// TIA Portal V18 export
FUNCTION_BLOCK "productionCounter"   // FB8, FBD
{ S7_Optimized_Access := 'TRUE' }
// stored: MemoryReserve 100, SetENOAutomatically false
   VAR_INPUT
      I_partProduced : Bool;
      I_nokPart : Bool;
   END_VAR
   VAR_IN_OUT
      IO_actualValues : "UDT_actualValues";
      IO_PreviousValues : "UDT_actualValues";
      IO_settings : "UDT_settings";
      IO_control : "UDT_control";
      IO_settingsShift1 : "UDT_settingsShift";
      IO_settingsShift2 : "UDT_settingsShift";
      IO_settingsShift3 : "UDT_settingsShift";
      IO_locTime : DTL;
   END_VAR
   VAR
      fpBit_resetCounters : Bool;
      fpBit_partProduced : Bool;
      fpBit_nokPart : Bool;
      fpBit_stop : Bool;
      fpBit_start : Bool;
      RS_taktTimeEn : Bool;
      TIM_taktTime { S7_SetPoint := 'True'} : TONR_TIME;
      memTaktTime : DInt;
      shiftTrigger0 { S7_SetPoint := 'True'} : "shiftTrigger";
      shiftTrigger1 { S7_SetPoint := 'True'} : "shiftTrigger";
      shiftTrigger2 { S7_SetPoint := 'True'} : "shiftTrigger";
      TaktTimeElapsed { S7_SetPoint := 'True'} : Time;
   END_VAR
   VAR_TEMP
      T_resetTaktTimeTimer : Bool;
      T_changeTaktTimeTimer : Bool;
      T_actualTOD : Time_Of_Day;
      T_shiftTrigger : Array[0..2] of Struct
         active : Bool;
         taktTimeEn : Bool;
         startDetect : Bool;
      END_STRUCT;
      T_control : Struct
         stop : Bool;
         start : Bool;
         resetCounters : Bool;
         taktTimeEn : Bool;
      END_STRUCT;
      T_settings : Struct
         enabled : Bool;
         autostartEnabled : Bool;
      END_STRUCT;
   END_VAR
   VAR_TEMP   // added for the SCL form of the ladder/FBD networks
      _w1 : Bool;
   END_VAR
BEGIN

REGION Network 1: free
END_REGION

REGION Network 2: actual TOD / Convert actual local time to TOD
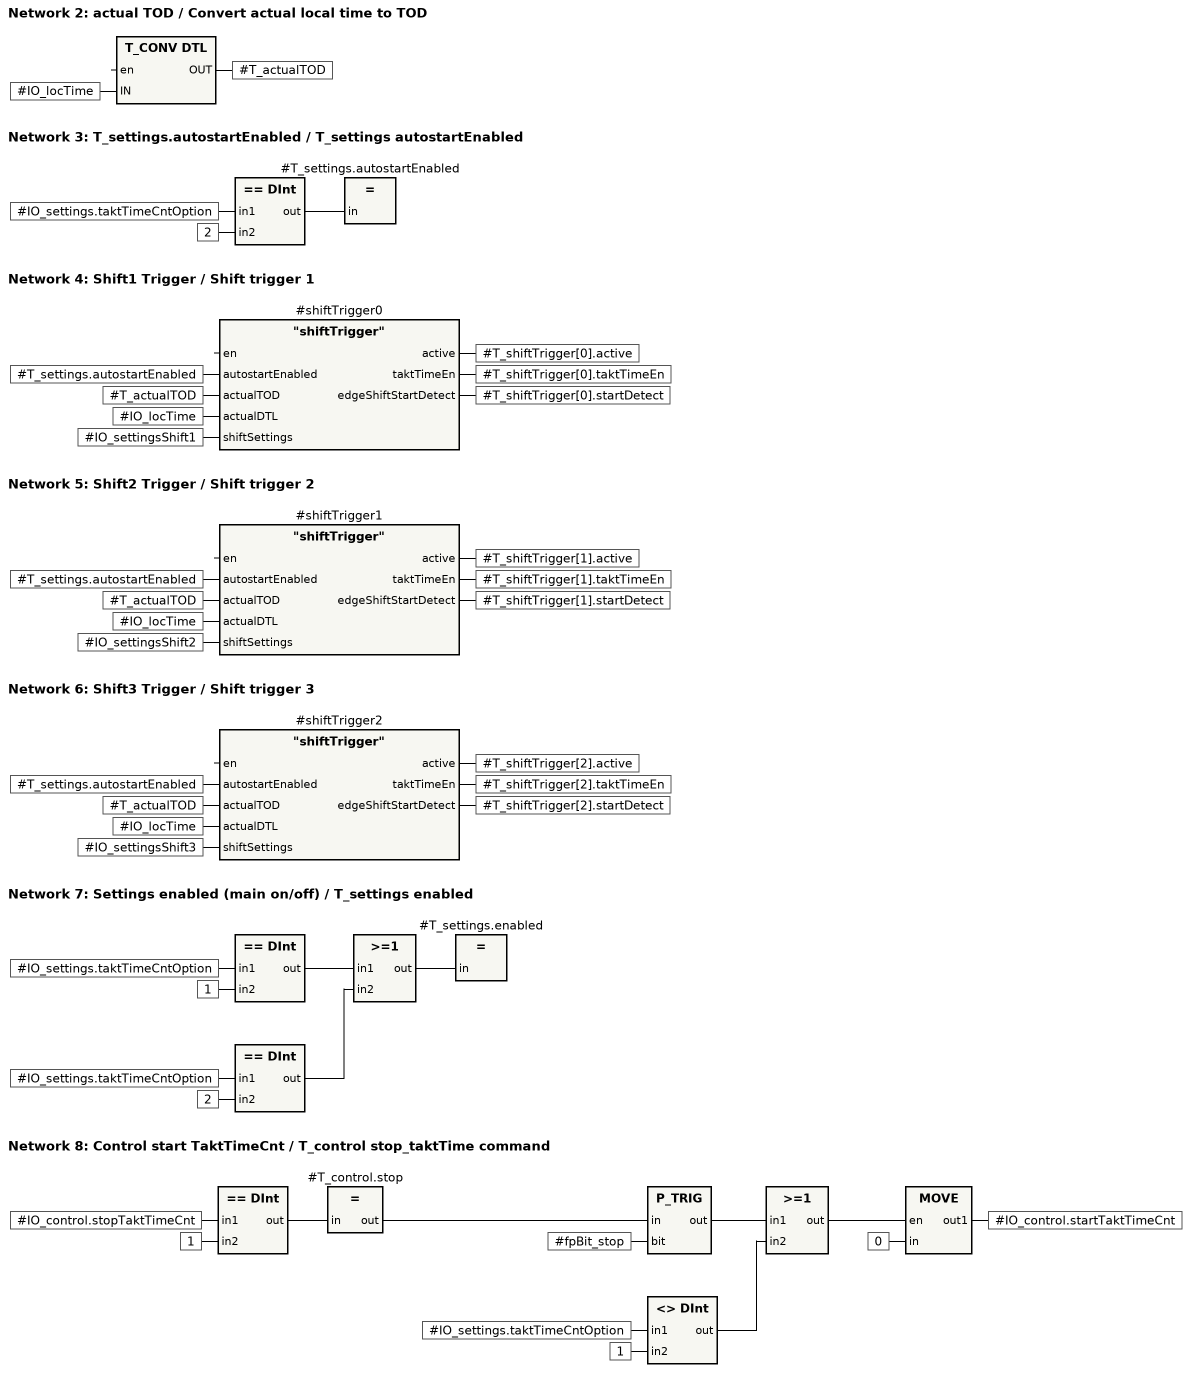
   T_CONV(IN := #IO_locTime, OUT => #T_actualTOD);
END_REGION

REGION Network 3: T_settings.autostartEnabled / T_settings autostartEnabled
   #T_settings.autostartEnabled := #IO_settings.taktTimeCntOption = 2;
END_REGION

REGION Network 4: Shift1 Trigger / Shift trigger 1
   #shiftTrigger0(autostartEnabled := #T_settings.autostartEnabled,   // "shiftTrigger"
                  actualTOD := #T_actualTOD,
                  actualDTL := #IO_locTime,
                  shiftSettings := #IO_settingsShift1,
                  active => #T_shiftTrigger[0].active,
                  taktTimeEn => #T_shiftTrigger[0].taktTimeEn,
                  edgeShiftStartDetect => #T_shiftTrigger[0].startDetect);
END_REGION

REGION Network 5: Shift2 Trigger / Shift trigger 2
   #shiftTrigger1(autostartEnabled := #T_settings.autostartEnabled,   // "shiftTrigger"
                  actualTOD := #T_actualTOD,
                  actualDTL := #IO_locTime,
                  shiftSettings := #IO_settingsShift2,
                  active => #T_shiftTrigger[1].active,
                  taktTimeEn => #T_shiftTrigger[1].taktTimeEn,
                  edgeShiftStartDetect => #T_shiftTrigger[1].startDetect);
END_REGION

REGION Network 6: Shift3 Trigger / Shift trigger 3
   #shiftTrigger2(autostartEnabled := #T_settings.autostartEnabled,   // "shiftTrigger"
                  actualTOD := #T_actualTOD,
                  actualDTL := #IO_locTime,
                  shiftSettings := #IO_settingsShift3,
                  active => #T_shiftTrigger[2].active,
                  taktTimeEn => #T_shiftTrigger[2].taktTimeEn,
                  edgeShiftStartDetect => #T_shiftTrigger[2].startDetect);
END_REGION

REGION Network 7: Settings enabled (main on/off) / T_settings enabled
   #T_settings.enabled := (#IO_settings.taktTimeCntOption = 1) OR (#IO_settings.taktTimeCntOption = 2);
END_REGION

REGION Network 8: Control start TaktTimeCnt / T_control stop_taktTime command
   #T_control.stop := #IO_control.stopTaktTimeCnt = 1;
   #_w1 := #T_control.stop AND NOT #fpBit_stop;   // rising edge
   #fpBit_stop := #T_control.stop;
   IF #_w1 OR (#IO_settings.taktTimeCntOption <> 1) THEN #IO_control.startTaktTimeCnt := 0; END_IF;
END_REGION

REGION Network 9: Control stop TaktTimeCnt / T_control start_taktTime command
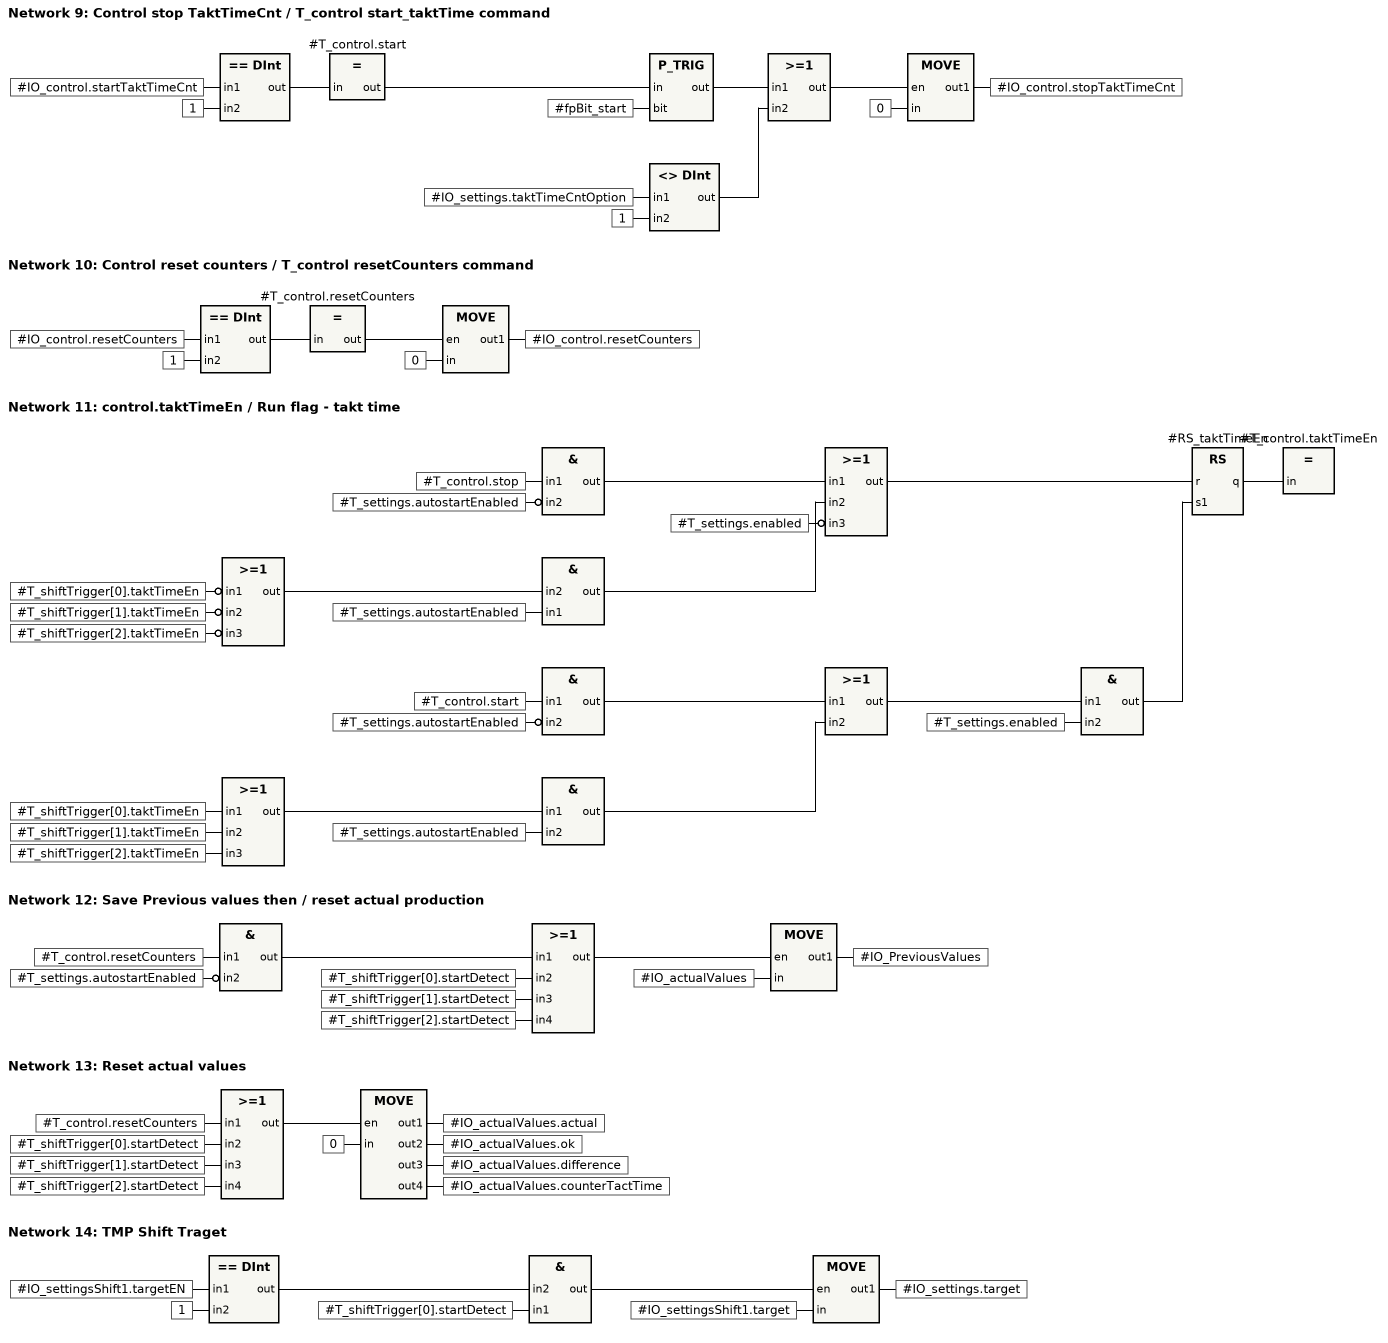
   #T_control.start := #IO_control.startTaktTimeCnt = 1;
   #_w1 := #T_control.start AND NOT #fpBit_start;   // rising edge
   #fpBit_start := #T_control.start;
   IF #_w1 OR (#IO_settings.taktTimeCntOption <> 1) THEN #IO_control.stopTaktTimeCnt := 0; END_IF;
END_REGION

REGION Network 10: Control reset counters / T_control resetCounters command
   #T_control.resetCounters := #IO_control.resetCounters = 1;
   IF #T_control.resetCounters THEN #IO_control.resetCounters := 0; END_IF;
END_REGION

REGION Network 11: control.taktTimeEn / Run flag - takt time
   IF (#T_control.stop AND NOT #T_settings.autostartEnabled) OR ((NOT #T_shiftTrigger[0].taktTimeEn OR NOT #T_shiftTrigger[1].taktTimeEn OR NOT #T_shiftTrigger[2].taktTimeEn) AND #T_settings.autostartEnabled) OR NOT #T_settings.enabled THEN
       #RS_taktTimeEn := FALSE;   // RS flip-flop
   END_IF;
   IF ((#T_control.start AND NOT #T_settings.autostartEnabled) OR ((#T_shiftTrigger[0].taktTimeEn OR #T_shiftTrigger[1].taktTimeEn OR #T_shiftTrigger[2].taktTimeEn) AND #T_settings.autostartEnabled)) AND #T_settings.enabled THEN
       #RS_taktTimeEn := TRUE;
   END_IF;
   #T_control.taktTimeEn := #RS_taktTimeEn;
END_REGION

REGION Network 12: Save Previous values then / reset actual production
   IF (#T_control.resetCounters AND NOT #T_settings.autostartEnabled) OR #T_shiftTrigger[0].startDetect OR #T_shiftTrigger[1].startDetect OR #T_shiftTrigger[2].startDetect THEN
       #IO_PreviousValues := #IO_actualValues;
   END_IF;
END_REGION

REGION Network 13: Reset actual values
   IF #T_control.resetCounters OR #T_shiftTrigger[0].startDetect OR #T_shiftTrigger[1].startDetect OR #T_shiftTrigger[2].startDetect THEN
       #IO_actualValues.actual := 0;
       #IO_actualValues.ok := 0;
       #IO_actualValues.difference := 0;
       #IO_actualValues.counterTactTime := 0;
   END_IF;
END_REGION

REGION Network 14: TMP Shift Traget
   IF (#IO_settingsShift1.targetEN = 1) AND #T_shiftTrigger[0].startDetect THEN
       #IO_settings.target := #IO_settingsShift1.target;
   END_IF;
END_REGION

REGION Network 15: #IO_settingsShift1.target - > #IO_settings.target
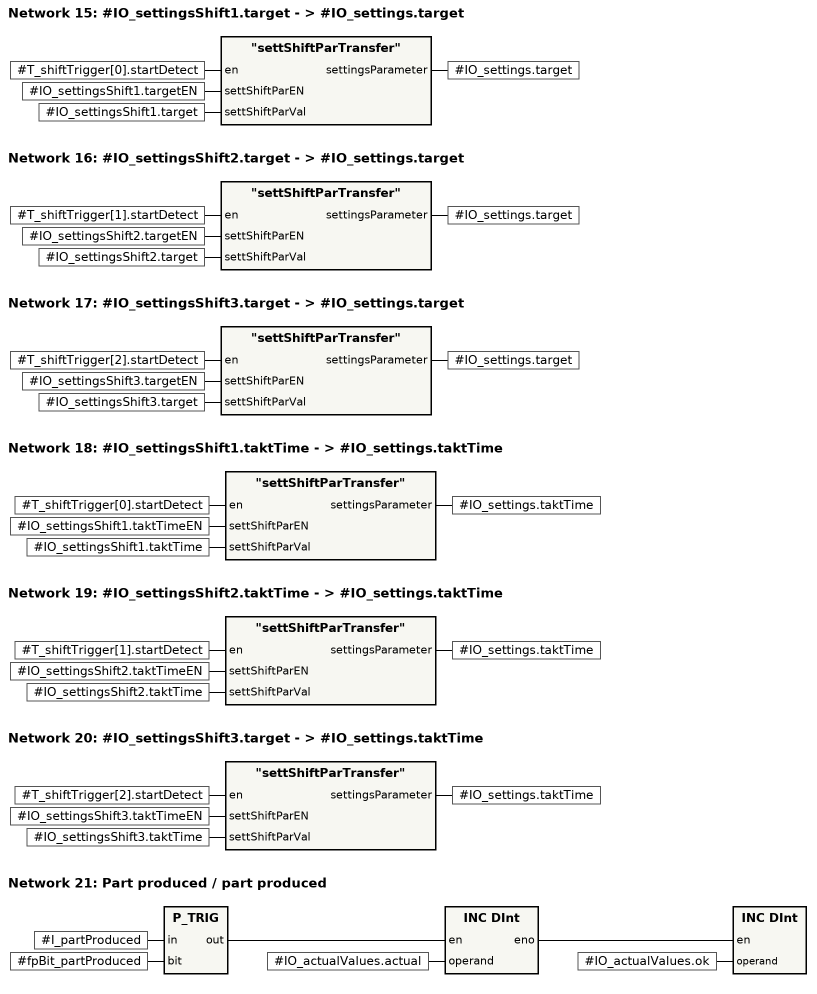
   IF #T_shiftTrigger[0].startDetect THEN
       "settShiftParTransfer"(settShiftParEN := #IO_settingsShift1.targetEN,
                              settShiftParVal := #IO_settingsShift1.target,
                              settingsParameter => #IO_settings.target);
   END_IF;
END_REGION

REGION Network 16: #IO_settingsShift2.target - > #IO_settings.target
   IF #T_shiftTrigger[1].startDetect THEN
       "settShiftParTransfer"(settShiftParEN := #IO_settingsShift2.targetEN,
                              settShiftParVal := #IO_settingsShift2.target,
                              settingsParameter => #IO_settings.target);
   END_IF;
END_REGION

REGION Network 17: #IO_settingsShift3.target - > #IO_settings.target
   IF #T_shiftTrigger[2].startDetect THEN
       "settShiftParTransfer"(settShiftParEN := #IO_settingsShift3.targetEN,
                              settShiftParVal := #IO_settingsShift3.target,
                              settingsParameter => #IO_settings.target);
   END_IF;
END_REGION

REGION Network 18: #IO_settingsShift1.taktTime - > #IO_settings.taktTime
   IF #T_shiftTrigger[0].startDetect THEN
       "settShiftParTransfer"(settShiftParEN := #IO_settingsShift1.taktTimeEN,
                              settShiftParVal := #IO_settingsShift1.taktTime,
                              settingsParameter => #IO_settings.taktTime);
   END_IF;
END_REGION

REGION Network 19: #IO_settingsShift2.taktTime - > #IO_settings.taktTime
   IF #T_shiftTrigger[1].startDetect THEN
       "settShiftParTransfer"(settShiftParEN := #IO_settingsShift2.taktTimeEN,
                              settShiftParVal := #IO_settingsShift2.taktTime,
                              settingsParameter => #IO_settings.taktTime);
   END_IF;
END_REGION

REGION Network 20: #IO_settingsShift3.target - > #IO_settings.taktTime
   IF #T_shiftTrigger[2].startDetect THEN
       "settShiftParTransfer"(settShiftParEN := #IO_settingsShift3.taktTimeEN,
                              settShiftParVal := #IO_settingsShift3.taktTime,
                              settingsParameter => #IO_settings.taktTime);
   END_IF;
END_REGION

REGION Network 21: Part produced / part produced
   // ENO of a box is taken as its EN; it also drops when the box reports an error
   #_w1 := #I_partProduced AND NOT #fpBit_partProduced;   // rising edge
   #fpBit_partProduced := #I_partProduced;
   IF #_w1 THEN
       #IO_actualValues.actual := #IO_actualValues.actual + 1;
       #IO_actualValues.ok := #IO_actualValues.ok + 1;
   END_IF;
END_REGION

REGION Network 22: Nok part / NOK part
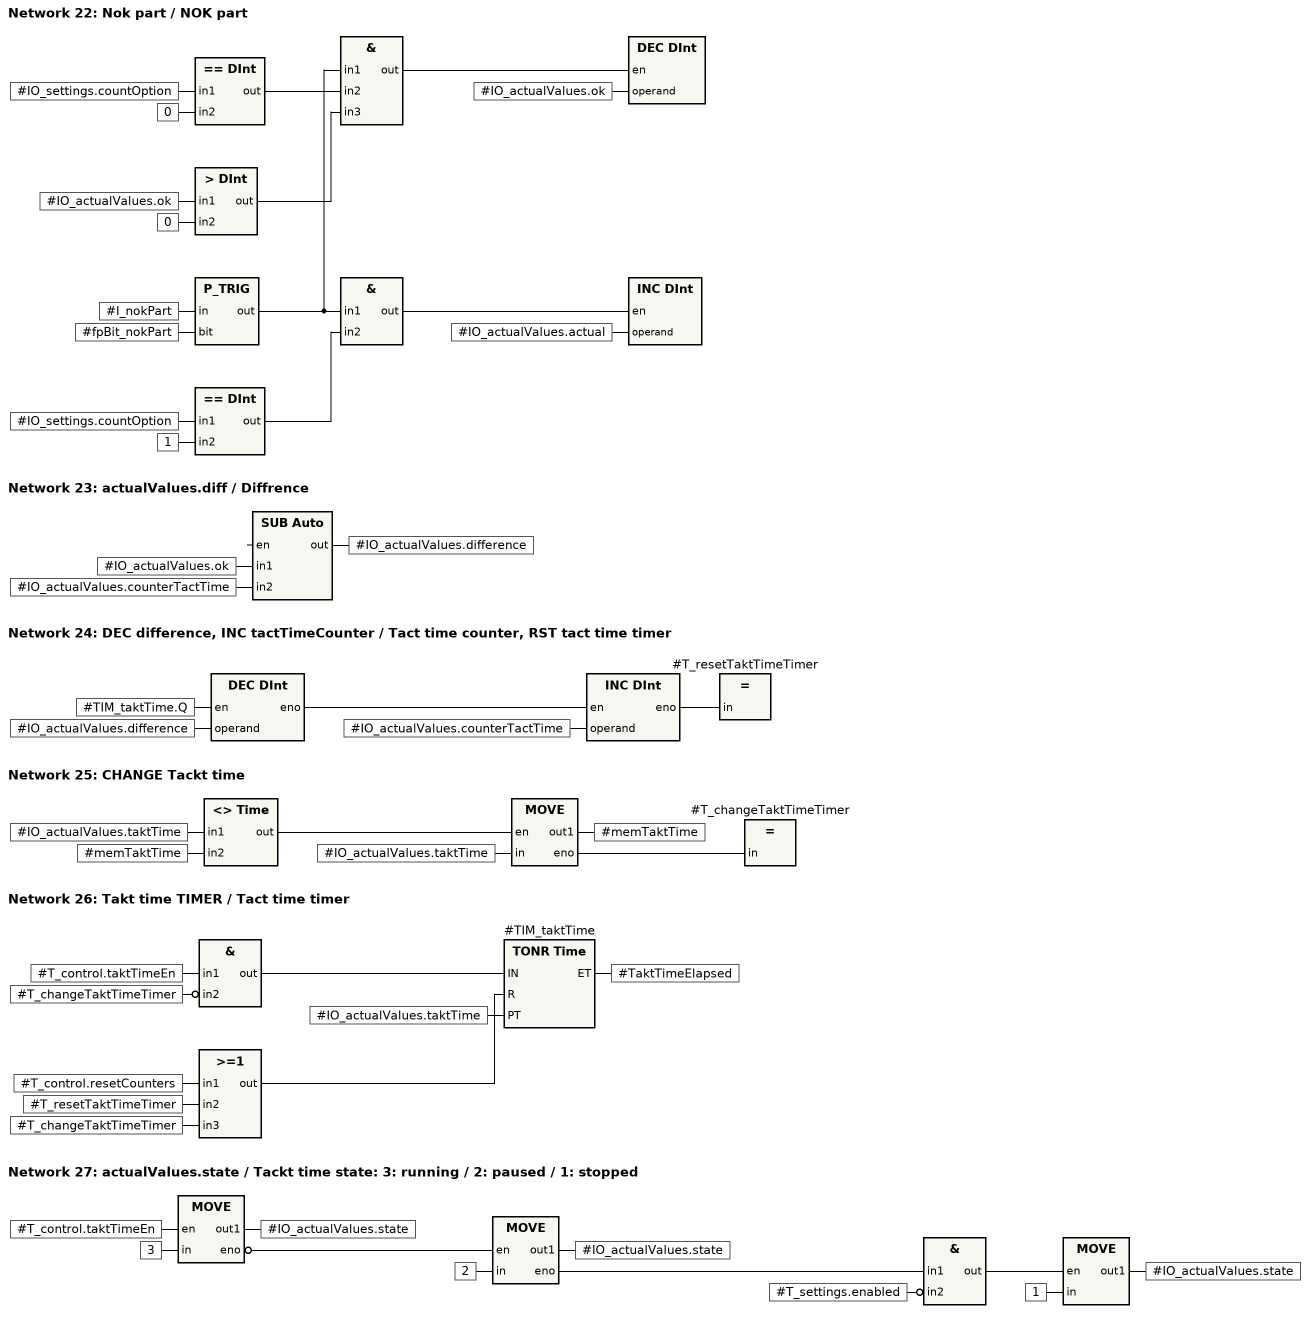
   #_w1 := #I_nokPart AND NOT #fpBit_nokPart;   // rising edge
   #fpBit_nokPart := #I_nokPart;
   IF #_w1 AND (#IO_settings.countOption = 0) AND (#IO_actualValues.ok > 0) THEN
       #IO_actualValues.ok := #IO_actualValues.ok - 1;
   END_IF;
   IF #_w1 AND (#IO_settings.countOption = 1) THEN
       #IO_actualValues.actual := #IO_actualValues.actual + 1;
   END_IF;
END_REGION

REGION Network 23: actualValues.diff / Diffrence
   #IO_actualValues.difference := #IO_actualValues.ok - #IO_actualValues.counterTactTime;
END_REGION

REGION Network 24: DEC difference, INC tactTimeCounter / Tact time counter, RST tact time timer
   // ENO of a box is taken as its EN; it also drops when the box reports an error
   IF #TIM_taktTime.Q THEN
       #IO_actualValues.difference := #IO_actualValues.difference - 1;
       #IO_actualValues.counterTactTime := #IO_actualValues.counterTactTime + 1;
   END_IF;
   #T_resetTaktTimeTimer := #TIM_taktTime.Q;
END_REGION

REGION Network 25: CHANGE Tackt time
   #_w1 := #IO_actualValues.taktTime <> #memTaktTime;
   IF #_w1 THEN #memTaktTime := #IO_actualValues.taktTime; END_IF;
   #T_changeTaktTimeTimer := #_w1;
END_REGION

REGION Network 26: Takt time TIMER / Tact time timer
   #TIM_taktTime(IN := #T_control.taktTimeEn AND NOT #T_changeTaktTimeTimer,   // TONR
                 R := #T_control.resetCounters OR #T_resetTaktTimeTimer OR #T_changeTaktTimeTimer,
                 PT := #IO_actualValues.taktTime,
                 ET => #TaktTimeElapsed);
END_REGION

REGION Network 27: actualValues.state / Tackt time state: 3: running / 2: paused / 1: stopped
   // ENO of a box is taken as its EN; it also drops when the box reports an error
   IF #T_control.taktTimeEn THEN #IO_actualValues.state := 3; END_IF;
   #_w1 := NOT #T_control.taktTimeEn;
   IF #_w1 THEN #IO_actualValues.state := 2; END_IF;
   IF #_w1 AND NOT #T_settings.enabled THEN #IO_actualValues.state := 1; END_IF;
END_REGION

REGION Network 28: settings.target -> actualValues.Target
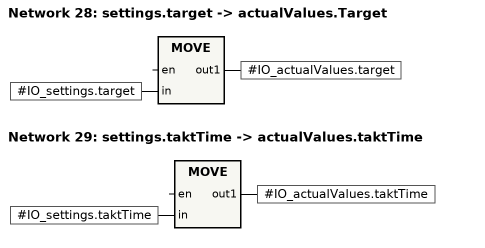
   #IO_actualValues.target := #IO_settings.target;
END_REGION

REGION Network 29: settings.taktTime -> actualValues.taktTime
   #IO_actualValues.taktTime := #IO_settings.taktTime;
END_REGION
END_FUNCTION_BLOCK
